// TIA Portal V20 export
// export: Created 2025-12-01T14:57:13.3807094Z, ExportSetting None, DisplayName Totally Integrated Automation Portal, DisplayVersion V20 Update 3, DisplayName TIA Portal Openness, DisplayVersion V20 Update 3, DisplayName TIA Portal Version Control Interface, DisplayVersion V20 Update 3, DisplayName STEP 7 Professional, DisplayVersion V20 Update 3, DisplayName STEP 7 Safety, DisplayVersion V20 Update 2, DisplayName WinCC Basic/Comfort/Advanced, DisplayVersion V20 Update 3, DisplayName WinCC Professional, DisplayVersion V20 Update 3, DisplayName WinCC Unified, DisplayVersion V20 Update 3
FUNCTION "FC884_BorrarError_Armarios" : Void   // FC884, LAD
{ S7_Optimized_Access := 'FALSE' }
AUTHOR : ERRORES
NAME : 20130301
VERSION : 3.0
// stored: AutoNumber false, SetENOAutomatically false
   VAR_INPUT
      NumDB_Errores : UInt;
      Numero : UInt;
   END_VAR
   VAR_IN_OUT
      Codigo : UDInt;
      Emergencia : Bool;
      ErrorGrave : Bool;
      ErrorLeve : Bool;
   END_VAR
   VAR_TEMP
      Guardar_AR1 : DWord;
      P_Inicial : DWord;
      P_Final : DWord;
      NumDB : Word;
      OffsetEmerg : UInt;
      OffsetErrorGrave : UInt;
      OffsetErrorLeve : UInt;
      MaxBitsGraves : UInt;
      MaxBitsLeves : UInt;
      LongBits : UInt;
      Zona : UInt;
   END_VAR
BEGIN

NETWORK
TITLE = Inicializar
///////////////////////////////////////////////////////////////////////////
// --- Inicializar Variables

      L     #NumDB_Errores;  // DB de Errores FIFO
      T     #NumDB;

      L     16;  // Long de la Estructura
      T     #LongBits;

      L     0;  // Offset de Los Bits
      T     #OffsetEmerg;
      L     2;
      T     #OffsetErrorGrave;
      L     4;
      T     #OffsetErrorLeve;

      L     15;  // Numero de Bits
      T     #MaxBitsGraves;
      L     95;
      T     #MaxBitsLeves;


      L     #Numero;
      T     #Zona;


///////////////////////////////////////////////////////////////////////////
// --- Comprobación del Numero de Dispositivo

      L     #Zona;
      L     0;
      <I;
      JC    Error_NumeroDispositivo;
      L     #Zona;
      L     "CTE_MaxDispositivos";
      >I;
      JC    Error_NumeroDispositivo;

      JU    Mirar_EmergenciaGrave;  // Ir a Mirar los Errores Graves



NETWORK
TITLE = Borrar el Array de Emergencias
Mirar_EmergenciaGrave:NOP   0;

///////////////////////////////////////////////////////////////////////////
// --- Preparar puntero Inicial y Final

      L     #Zona;
      L     #LongBits;
      *D;
      L     #OffsetEmerg;
      +D;
      SLD   3;
      T     #P_Inicial;
      T     #P_Final;


///////////////////////////////////////////////////////////////////////////
// --- Recorrer el Arrray, para resetear los Bits

Bucle_EmergenciaGrave:NOP   0;
      OPN   DB [#NumDB];  // Recorrer todos los Bits
      SET;
      R     DBX [#P_Final];

      L     #P_Final;
      L     #P_Inicial;
      -D;
      L     #MaxBitsGraves;
      ==I;
      JC    Mirar_ErrorGrave;  // Si ha recorrido todos los bits

      L     #P_Final;
      L     P#0.1;
      +D;
      T     #P_Final;
      JU    Bucle_EmergenciaGrave;  // Siguiente Bit



NETWORK
TITLE = Borrar el Array de Errorres de Graves
Mirar_ErrorGrave:NOP   0;

///////////////////////////////////////////////////////////////////////////
// --- Preparar puntero Inicial y Final

      L     #Zona;
      L     #LongBits;
      *D;
      L     #OffsetErrorGrave;
      +D;
      SLD   3;
      T     #P_Inicial;
      T     #P_Final;


///////////////////////////////////////////////////////////////////////////
// --- Recorrer el arrray, para resetear los Bits

Bucle_ErrorGrave:NOP   0;
      OPN   DB [#NumDB];  // Recorrer todos los Bits
      SET;
      R     DBX [#P_Final];

      L     #P_Final;
      L     #P_Inicial;
      -D;
      L     #MaxBitsGraves;
      ==I;
      JC    Mirar_ErrorLeve;  // Si ha recorrido todos los bits

      L     #P_Final;
      L     P#0.1;
      +D;
      T     #P_Final;
      JU    Bucle_ErrorGrave;  // Siguiente Bit



NETWORK
TITLE = Borrar el Array de Errores de Leves
Mirar_ErrorLeve:NOP   0;

///////////////////////////////////////////////////////////////////////////
// --- Preparar puntero Inicial y Final

      L     #Zona;
      L     #LongBits;
      *D;
      L     #OffsetErrorLeve;
      +D;
      SLD   3;
      T     #P_Inicial;
      T     #P_Final;


///////////////////////////////////////////////////////////////////////////
// --- Recorrer el arrray, para resetear los Bits

Bucle_ErrorLeve:NOP   0;
      OPN   DB [#NumDB];  // Recorrer todos los bits
      SET;
      R     DBX [#P_Final];

      L     #P_Final;
      L     #P_Inicial;
      -D;
      L     #MaxBitsLeves;
      ==I;
      JC    Final;  // Si ha recorrido todos los bits

      L     #P_Final;
      L     P#0.1;
      +D;
      T     #P_Final;
      JU    Bucle_ErrorLeve;  // Siguiente Bit



NETWORK
TITLE = Finalizar
Final:NOP   0;

///////////////////////////////////////////////////////////////////////////
// --- Salida de la Funcion:
// ---      Escribir el Error
// ---      Preparar para Visualizar
// ---      Resetear los Bits Graves y Leves

      L     0;
      T     #Codigo;

      T     "DB861_FIFO_Errores".ArmariosGraves[#Zona];
      T     "DB861_FIFO_Errores".ArmariosLeves[#Zona];

      SET;
      R     #Emergencia;
      R     #ErrorGrave;
      R     #ErrorLeve;


///////////////////////////////////////////////////////////////////////////
// --- Se acabo la Funcion

Error_NumeroDispositivo:NOP   0;



END_FUNCTION
